// TIA Portal V20 export
FUNCTION_BLOCK "LER_Axis_Absolute"   // FB186, LAD
// stored: Access Published, MemoryReserve 100, SetENOAutomatically false
   VAR_INPUT
      PosiNo : SInt;
      Status : "LAF_typeUnitStatus";
      int1 { ExternalAccessible := 'False'; ExternalVisible := 'False'; ExternalWritable := 'False'} : Bool := FALSE;
      int2 { ExternalAccessible := 'False'; ExternalVisible := 'False'; ExternalWritable := 'False'} : Bool := TRUE;
      int3 { ExternalAccessible := 'False'; ExternalVisible := 'False'; ExternalWritable := 'False'} : Bool := TRUE;
      int4 { ExternalAccessible := 'False'; ExternalVisible := 'False'; ExternalWritable := 'False'} : Bool := TRUE;
      int5 { ExternalAccessible := 'False'; ExternalVisible := 'False'; ExternalWritable := 'False'} : Bool := TRUE;
      int6 { ExternalAccessible := 'False'; ExternalVisible := 'False'; ExternalWritable := 'False'} : Bool := TRUE;
      int7 { ExternalAccessible := 'False'; ExternalVisible := 'False'; ExternalWritable := 'False'} : Bool := TRUE;
      int8 { ExternalAccessible := 'False'; ExternalVisible := 'False'; ExternalWritable := 'False'} : Bool := TRUE;
      int9 { ExternalAccessible := 'False'; ExternalVisible := 'False'; ExternalWritable := 'False'} : Bool := TRUE;
      int10 { ExternalAccessible := 'False'; ExternalVisible := 'False'; ExternalWritable := 'False'} : Bool := TRUE;
      Bypass : Bool := FALSE;
      commands : "LBC_typeAxis64PosManualCommands";
   END_VAR
   VAR_IN_OUT
      interlockOk : Array[0..15] of Bool;
      intOut : Array[0..9] of Bool;
   END_VAR
   VAR
      "Condition Run" { ExternalVisible := 'False'} : Bool;
      condition : Bool;
      NotCondition { ExternalVisible := 'False'} : Bool;
      point { ExternalVisible := 'False'} : SInt;
   END_VAR
BEGIN

REGION Network 1
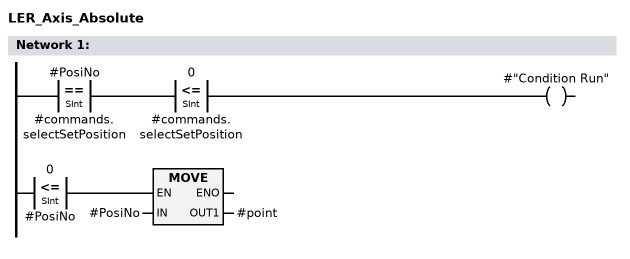
   RUNG wire#powerrail
      { S7_Templates := "SrcType := SInt" } EQ_Contact(in1 := #PosiNo, in2 := #commands.selectSetPosition)
      { S7_Templates := "SrcType := SInt" } LE_Contact(in1 := 0, in2 := #commands.selectSetPosition)
      Coil( #"Condition Run" )
   END_RUNG
   RUNG wire#powerrail
      { S7_Templates := "SrcType := SInt" } LE_Contact(in1 := 0, in2 := #PosiNo)
      Move(in := #PosiNo, out1 => #point)
   END_RUNG
   // the same network as SCL:
   #"Condition Run" := (#PosiNo = #commands.selectSetPosition) AND (0 <= #commands.selectSetPosition);
   IF 0 <= #PosiNo THEN #point := #PosiNo; END_IF;
END_REGION

REGION Network 2 (SCL)



   IF (#int1 AND #int2 AND #int3 AND #int4 AND #int5 AND #int6 AND #int7 AND #int8 AND #int9 AND #int10 )OR #Bypass THEN
       #condition := TRUE;
       #NotCondition := FALSE;

       IF #"Condition Run" THEN
           #intOut[0] := FALSE;
           #intOut[1] := FALSE;
           #intOut[2] := FALSE;
           #intOut[3] := FALSE;
           #intOut[4] := FALSE;
           #intOut[5] := FALSE;
           #intOut[6] := FALSE;
           #intOut[7] := FALSE;
           #intOut[8] := FALSE;
           #intOut[9] := FALSE;
       END_IF;

   ELSE
        #condition := FALSE;
        #NotCondition := TRUE;

        IF #"Condition Run" THEN
            IF NOT #int1 THEN
                #intOut[0] := TRUE;
            ELSE
                #intOut[0] := FALSE;
            END_IF;
            IF NOT #int2 THEN
                #intOut[1] := TRUE;
            ELSE
                #intOut[1] := FALSE;
            END_IF;
            IF NOT #int3 THEN
                #intOut[2] := TRUE;
            ELSE
                #intOut[2] := FALSE;
            END_IF;
            IF NOT #int4 THEN
                #intOut[3] := TRUE;
            ELSE
                #intOut[3] := FALSE;
            END_IF;
            IF NOT #int5 THEN
                #intOut[4] := TRUE;
            ELSE
                #intOut[4] := FALSE;
            END_IF;
            IF NOT #int6 THEN
                #intOut[5] := TRUE;
            ELSE
                #intOut[5] := FALSE;
            END_IF;
            IF NOT #int7 THEN
                #intOut[6] := TRUE;
            ELSE
                #intOut[6] := FALSE;
            END_IF;
            IF NOT #int8 THEN
                #intOut[7] := TRUE;
            ELSE
                #intOut[7] := FALSE;
            END_IF;
            IF NOT #int9 THEN
                #intOut[8] := TRUE;
            ELSE
                #intOut[8] := FALSE;
            END_IF;
            IF NOT #int10 THEN
                #intOut[9] := TRUE;
            ELSE
                #intOut[9] := FALSE;
            END_IF;
        END_IF;
    END_IF;
    #interlockOk[#point] := #condition;
END_REGION
END_FUNCTION_BLOCK
